FUNCTION_BLOCK PierToPierCFB (* Composite Function Block Type *)
  (* Standard: 61499-2 *)
  (* Version 0.0, 2011-03-19, Majid Sorouri, nxtControl GmbH, template *)
  (* Compiler header: package fb.rt.pnp; *)
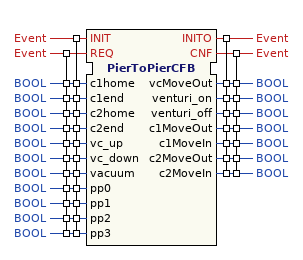
  EVENT_INPUT
    INIT WITH c1home, c1end, c2home, c2end, vc_up, vc_down, vacuum, pp0, pp1, pp2, pp3; (* Initialization Request *)
    REQ WITH c1home, c1end, c2home, c2end, vc_up, vc_down, vacuum, pp0, pp1, pp2, pp3; (* Normal Execution Request *)
  END_EVENT
  EVENT_OUTPUT
    INITO WITH venturi_off, vcMoveOut, venturi_on, c1MoveOut, c1MoveIn, c2MoveOut, c2MoveIn; (* Initialization Confirm *)
    CNF WITH vcMoveOut, venturi_on, venturi_off, c1MoveOut, c1MoveIn, c2MoveOut, c2MoveIn; (* Execution Confirmation *)
  END_EVENT
  VAR_INPUT
    c1home : BOOL;
    c1end : BOOL;
    c2home : BOOL;
    c2end : BOOL;
    vc_up : BOOL;
    vc_down : BOOL;
    vacuum : BOOL;
    pp0 : BOOL;
    pp1 : BOOL;
    pp2 : BOOL;
    pp3 : BOOL;
  END_VAR
  VAR_OUTPUT
    vcMoveOut : BOOL;
    venturi_on : BOOL;
    venturi_off : BOOL;
    c1MoveOut : BOOL;
    c1MoveIn : BOOL;
    c2MoveOut : BOOL;
    c2MoveIn : BOOL;
  END_VAR
  FBS
    FB3 : vaccum3;
    FB5 : E_Split4;
    FB2 : GenCyl(ID := 2);
    FB1 : GenCyl(ID := 1);
    FB4 : verticalcylinder3;
    FB6 : E_SPLIT;
  END_FBS
  EVENT_CONNECTIONS
    INIT TO FB1.INIT;
    FB1.INITO TO FB2.INIT;
    FB2.INITO TO FB4.INIT;
    FB4.INITO TO FB3.INIT;
    REQ TO FB5.E;
    FB5.E1 TO FB1.REQ;
    FB5.E2 TO FB2.REQ;
    FB5.E3 TO FB4.REQ;
    FB5.E4 TO FB3.Req;
    FB4.OUT_CMD2 TO FB6.EI;
    FB6.EO2 TO FB1.IN_CMD;
    FB6.EO1 TO FB2.IN_CMD;
    FB2.OUT_CMD TO FB4.IN_CMD;
    FB3.OUT_CMD TO FB4.IN_CMD;
    FB1.OUT_CMD TO FB4.IN_CMD;
    FB4.OUT_CMD TO FB3.IN_CMD;
    FB3.INITO TO INITO;
    FB1.CNF TO CNF;
    FB2.CNF TO CNF;
    FB4.CNF TO CNF;
    FB3.CNF TO CNF;
  END_CONNECTIONS
  DATA_CONNECTIONS
    FB4.DownToPick TO FB3.SwitchOn;
    FB4.DownToDrop TO FB3.SwitchOff;
    FB1.AllowVcDown TO FB4.c1permitDown;
    FB2.AllowVcDown TO FB4.c2PermitDown;
    FB4.vc_Done TO FB2.vcPermitMove;
    FB4.vc_Done TO FB1.vcPermitMove;
    pp1 TO FB1.pp1;
    pp2 TO FB1.pp2;
    pp3 TO FB1.pp3;
    pp1 TO FB2.pp1;
    pp2 TO FB2.pp2;
    pp3 TO FB2.pp3;
    pp0 TO FB4.pp0;
    vc_up TO FB4.vc_up;
    vc_down TO FB4.vc_down;
    c1home TO FB4.c1home;
    c2home TO FB4.c2home;
    FB4.vcMoveOut TO vcMoveOut;
    vacuum TO FB3.vacuum;
    FB3.venturi_on TO venturi_on;
    FB3.venturi_off TO venturi_off;
    c1home TO FB1.chome;
    c1end TO FB1.cend;
    c2home TO FB2.chome;
    c2end TO FB2.cend;
    FB1.cMoveOut TO c1MoveOut;
    FB1.cMoveIn TO c1MoveIn;
    FB2.cMoveOut TO c2MoveOut;
    FB2.cMoveIn TO c2MoveIn;
  END_CONNECTIONS
END_FUNCTION_BLOCK
